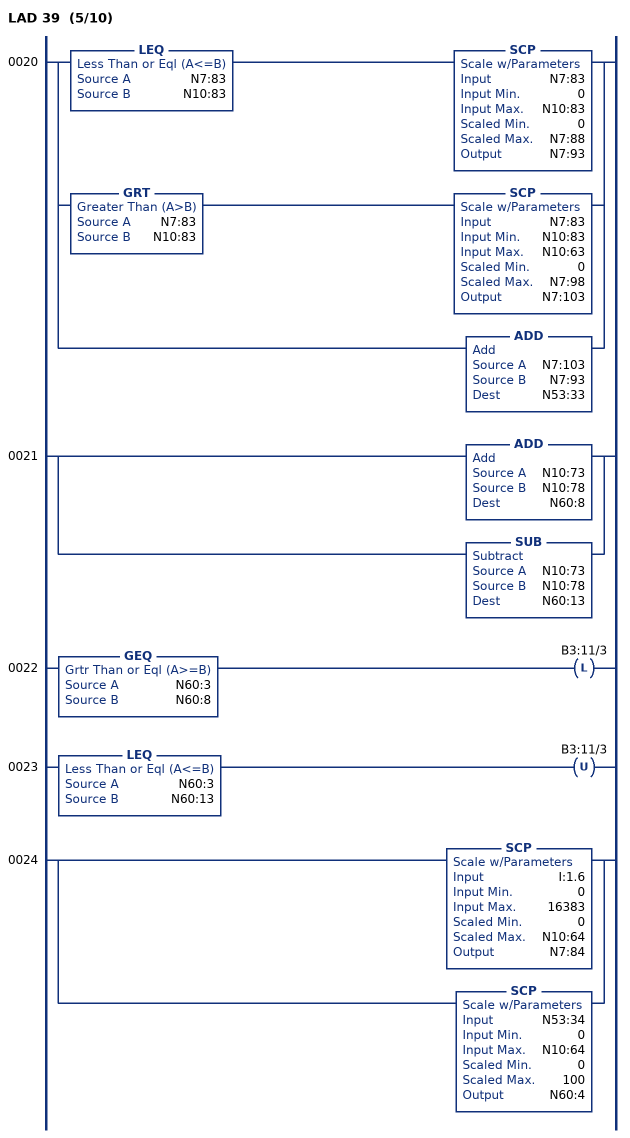
% Rung: 20 %
SOR BST LEQ N7:83 N10:83 SCP N7:83 0 N10:83 0 N7:88 N7:93 NXB GRT N7:83 N10:83 SCP N7:83 N10:83 N10:63 0 N7:98 N7:103 NXB ADD N7:103 N7:93 N53:33 BND EOR
% Rung: 21 %
SOR BST ADD N10:73 N10:78 N60:8 NXB SUB N10:73 N10:78 N60:13 BND EOR
% Rung: 22 %
SOR GEQ N60:3 N60:8 OTL B3:11/3 EOR
% Rung: 23 %
SOR LEQ N60:3 N60:13 OTU B3:11/3 EOR
% Rung: 24 %
SOR BST SCP I:1.6 0 16383 0 N10:64 N7:84 NXB SCP N53:34 0 N10:64 0 100 N60:4 BND EOR

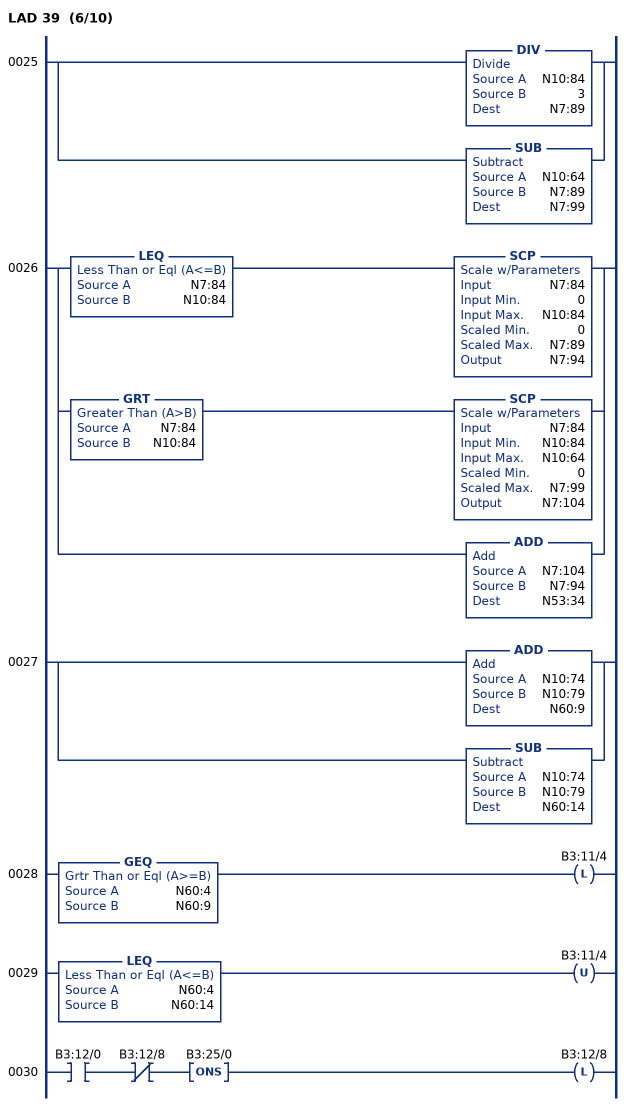
% Rung: 25 %
SOR BST DIV N10:84 3 N7:89 NXB SUB N10:64 N7:89 N7:99 BND EOR
% Rung: 26 %
SOR BST LEQ N7:84 N10:84 SCP N7:84 0 N10:84 0 N7:89 N7:94 NXB GRT N7:84 N10:84 SCP N7:84 N10:84 N10:64 0 N7:99 N7:104 NXB ADD N7:104 N7:94 N53:34 BND EOR
% Rung: 27 %
SOR BST ADD N10:74 N10:79 N60:9 NXB SUB N10:74 N10:79 N60:14 BND EOR
% Rung: 28 %
SOR GEQ N60:4 N60:9 OTL B3:11/4 EOR
% Rung: 29 %
SOR LEQ N60:4 N60:14 OTU B3:11/4 EOR
% Rung: 30 %
SOR XIC B3:12/0 XIO B3:12/8 OSR B3:25/0 OTL B3:12/8 EOR

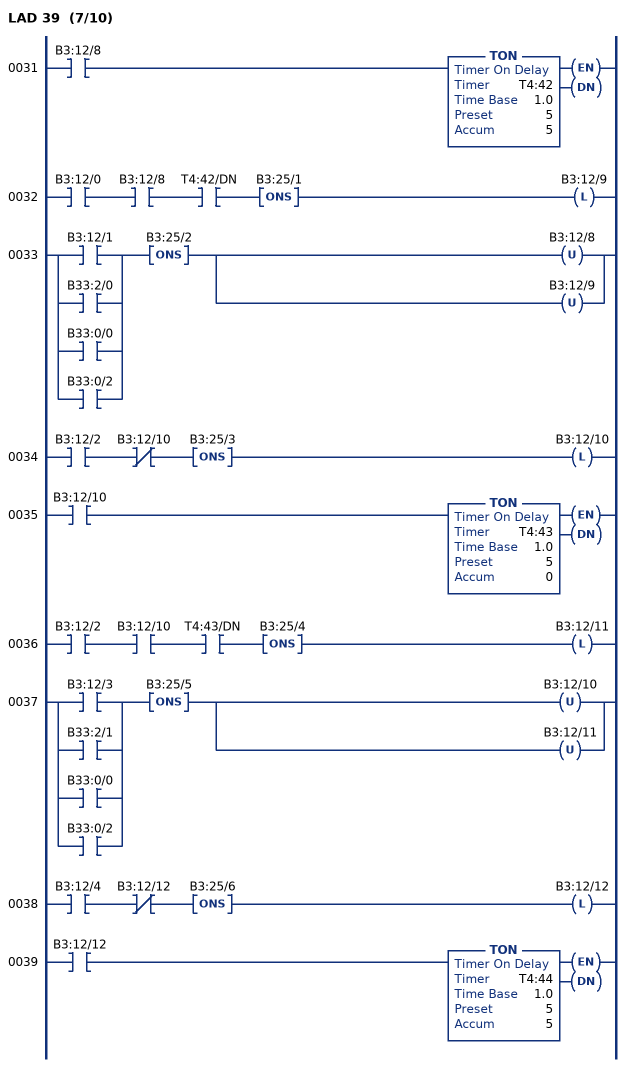
% Rung: 31 %
SOR XIC B3:12/8 TON T4:42 1.0 5 5 EOR
% Rung: 32 %
SOR XIC B3:12/0 XIC B3:12/8 XIC T4:42/DN OSR B3:25/1 OTL B3:12/9 EOR
% Rung: 33 %
SOR BST XIC B3:12/1 NXB XIC B33:2/0 NXB XIC B33:0/0 NXB XIC B33:0/2 BND OSR B3:25/2 BST OTU B3:12/8 NXB OTU B3:12/9 BND EOR
% Rung: 34 %
SOR XIC B3:12/2 XIO B3:12/10 OSR B3:25/3 OTL B3:12/10 EOR
% Rung: 35 %
SOR XIC B3:12/10 TON T4:43 1.0 5 0 EOR
% Rung: 36 %
SOR XIC B3:12/2 XIC B3:12/10 XIC T4:43/DN OSR B3:25/4 OTL B3:12/11 EOR
% Rung: 37 %
SOR BST XIC B3:12/3 NXB XIC B33:2/1 NXB XIC B33:0/0 NXB XIC B33:0/2 BND OSR B3:25/5 BST OTU B3:12/10 NXB OTU B3:12/11 BND EOR
% Rung: 38 %
SOR XIC B3:12/4 XIO B3:12/12 OSR B3:25/6 OTL B3:12/12 EOR
% Rung: 39 %
SOR XIC B3:12/12 TON T4:44 1.0 5 5 EOR

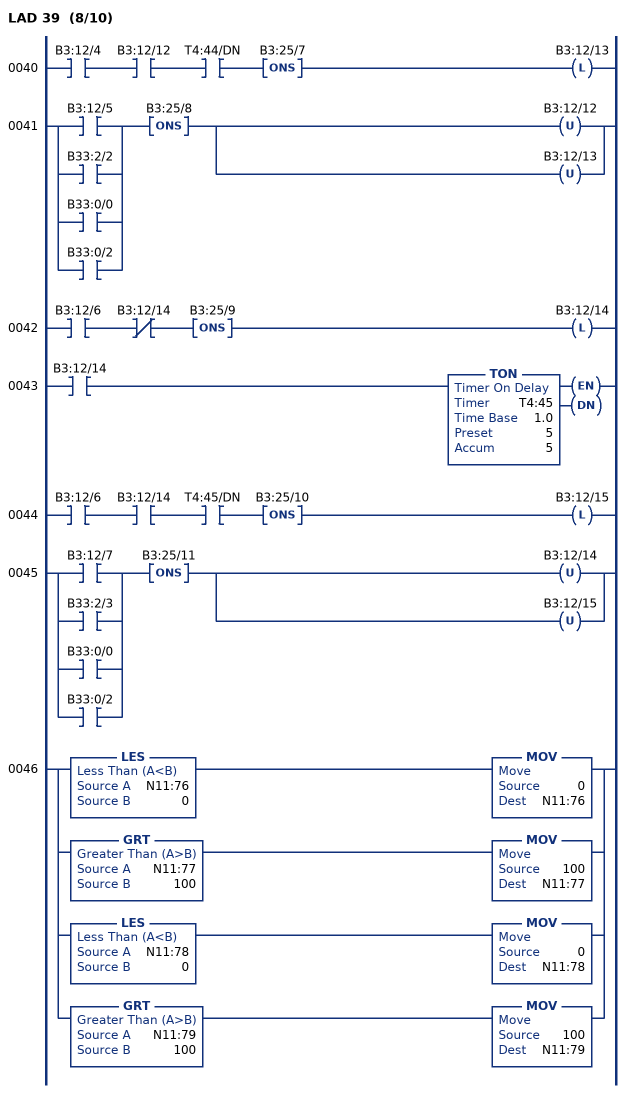
% Rung: 40 %
SOR XIC B3:12/4 XIC B3:12/12 XIC T4:44/DN OSR B3:25/7 OTL B3:12/13 EOR
% Rung: 41 %
SOR BST XIC B3:12/5 NXB XIC B33:2/2 NXB XIC B33:0/0 NXB XIC B33:0/2 BND OSR B3:25/8 BST OTU B3:12/12 NXB OTU B3:12/13 BND EOR
% Rung: 42 %
SOR XIC B3:12/6 XIO B3:12/14 OSR B3:25/9 OTL B3:12/14 EOR
% Rung: 43 %
SOR XIC B3:12/14 TON T4:45 1.0 5 5 EOR
% Rung: 44 %
SOR XIC B3:12/6 XIC B3:12/14 XIC T4:45/DN OSR B3:25/10 OTL B3:12/15 EOR
% Rung: 45 %
SOR BST XIC B3:12/7 NXB XIC B33:2/3 NXB XIC B33:0/0 NXB XIC B33:0/2 BND OSR B3:25/11 BST OTU B3:12/14 NXB OTU B3:12/15 BND EOR
% Rung: 46 %
SOR BST LES N11:76 0 MOV 0 N11:76 NXB GRT N11:77 100 MOV 100 N11:77 NXB LES N11:78 0 MOV 0 N11:78 NXB GRT N11:79 100 MOV 100 N11:79 BND EOR

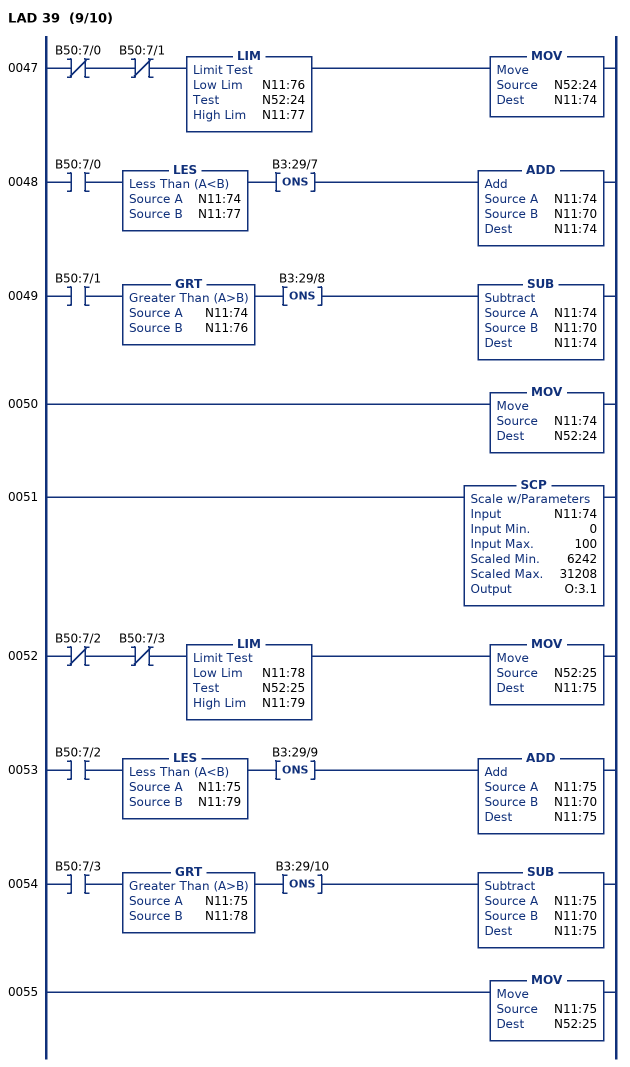
% Rung: 47 %
SOR XIO B50:7/0 XIO B50:7/1 LIM N11:76 N52:24 N11:77 MOV N52:24 N11:74 EOR
% Rung: 48 %
SOR XIC B50:7/0 LES N11:74 N11:77 OSR B3:29/7 ADD N11:74 N11:70 N11:74 EOR
% Rung: 49 %
SOR XIC B50:7/1 GRT N11:74 N11:76 OSR B3:29/8 SUB N11:74 N11:70 N11:74 EOR
% Rung: 50 %
SOR MOV N11:74 N52:24 EOR
% Rung: 51 %
SOR SCP N11:74 0 100 6242 31208 O:3.1 EOR
% Rung: 52 %
SOR XIO B50:7/2 XIO B50:7/3 LIM N11:78 N52:25 N11:79 MOV N52:25 N11:75 EOR
% Rung: 53 %
SOR XIC B50:7/2 LES N11:75 N11:79 OSR B3:29/9 ADD N11:75 N11:70 N11:75 EOR
% Rung: 54 %
SOR XIC B50:7/3 GRT N11:75 N11:78 OSR B3:29/10 SUB N11:75 N11:70 N11:75 EOR
% Rung: 55 %
SOR MOV N11:75 N52:25 EOR

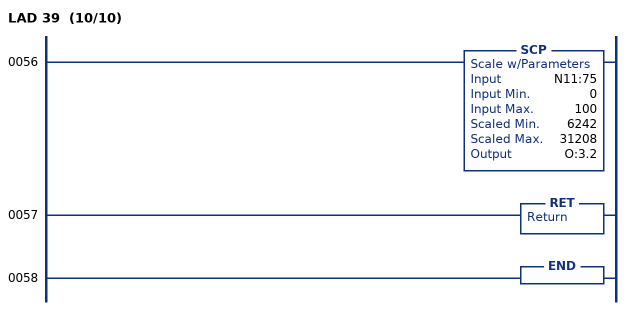
% Rung: 56 %
SOR SCP N11:75 0 100 6242 31208 O:3.2 EOR
% Rung: 57 %
SOR RET EOR
% Rung: 58 %
SOR END EOR

LADDER 40
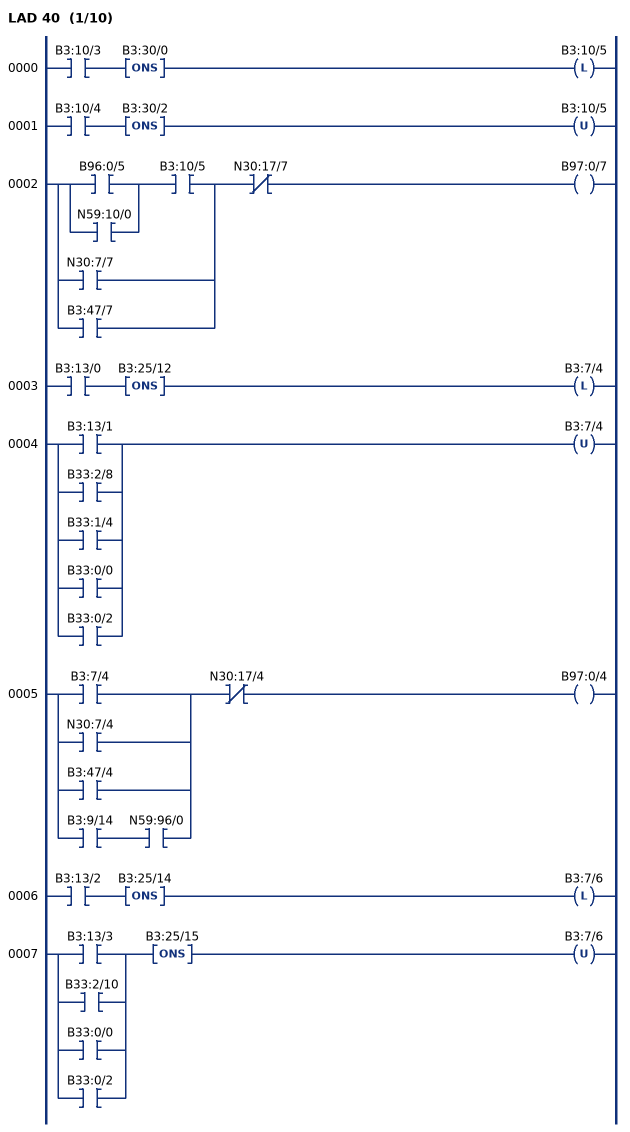
% Rung: 0 %
SOR XIC B3:10/3 OSR B3:30/0 OTL B3:10/5 EOR
% Rung: 1 %
SOR XIC B3:10/4 OSR B3:30/2 OTU B3:10/5 EOR
% Rung: 2 %
SOR BST BST XIC B96:0/5 NXB XIC N59:10/0 BND XIC B3:10/5 NXB XIC N30:7/7 NXB XIC B3:47/7 BND XIO N30:17/7 OTE B97:0/7 EOR
% Rung: 3 %
SOR XIC B3:13/0 OSR B3:25/12 OTL B3:7/4 EOR
% Rung: 4 %
SOR BST XIC B3:13/1 NXB XIC B33:2/8 NXB XIC B33:1/4 NXB XIC B33:0/0 NXB XIC B33:0/2 BND OTU B3:7/4 EOR
% Rung: 5 %
SOR BST XIC B3:7/4 NXB XIC N30:7/4 NXB XIC B3:47/4 NXB XIC B3:9/14 XIC N59:96/0 BND XIO N30:17/4 OTE B97:0/4 EOR
% Rung: 6 %
SOR XIC B3:13/2 OSR B3:25/14 OTL B3:7/6 EOR
% Rung: 7 %
SOR BST XIC B3:13/3 NXB XIC B33:2/10 NXB XIC B33:0/0 NXB XIC B33:0/2 BND OSR B3:25/15 OTU B3:7/6 EOR

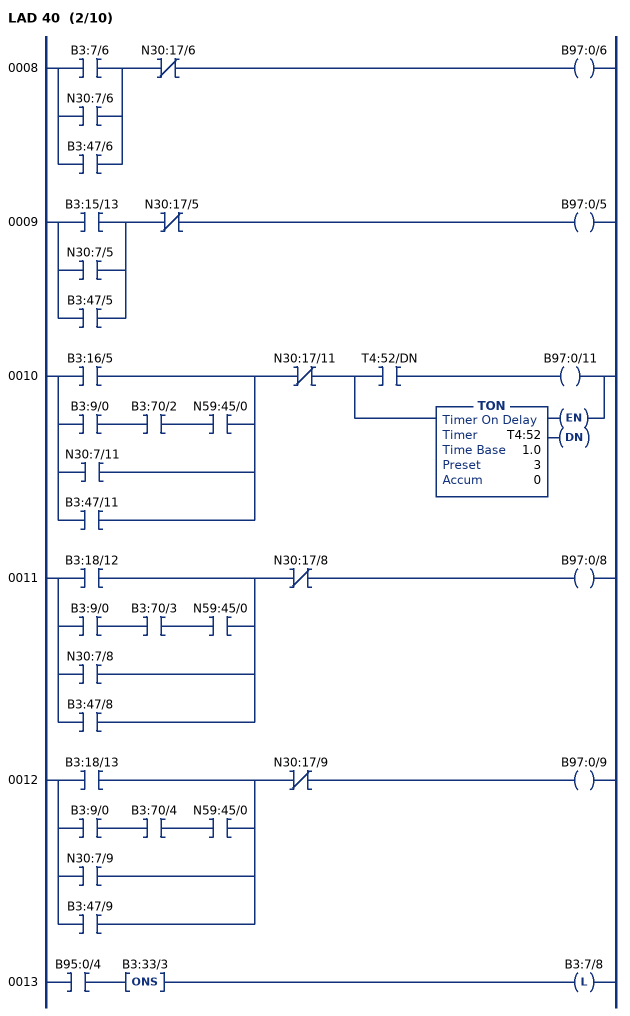
% Rung: 8 %
SOR BST XIC B3:7/6 NXB XIC N30:7/6 NXB XIC B3:47/6 BND XIO N30:17/6 OTE B97:0/6 EOR
% Rung: 9 %
SOR BST XIC B3:15/13 NXB XIC N30:7/5 NXB XIC B3:47/5 BND XIO N30:17/5 OTE B97:0/5 EOR
% Rung: 10 %
SOR BST XIC B3:16/5 NXB XIC B3:9/0 XIC B3:70/2 XIC N59:45/0 NXB XIC N30:7/11 NXB XIC B3:47/11 BND XIO N30:17/11 BST XIC T4:52/DN OTE B97:0/11 NXB TON T4:52 1.0 3 0 BND EOR
% Rung: 11 %
SOR BST XIC B3:18/12 NXB XIC B3:9/0 XIC B3:70/3 XIC N59:45/0 NXB XIC N30:7/8 NXB XIC B3:47/8 BND XIO N30:17/8 OTE B97:0/8 EOR
% Rung: 12 %
SOR BST XIC B3:18/13 NXB XIC B3:9/0 XIC B3:70/4 XIC N59:45/0 NXB XIC N30:7/9 NXB XIC B3:47/9 BND XIO N30:17/9 OTE B97:0/9 EOR
% Rung: 13 %
SOR XIC B95:0/4 OSR B3:33/3 OTL B3:7/8 EOR

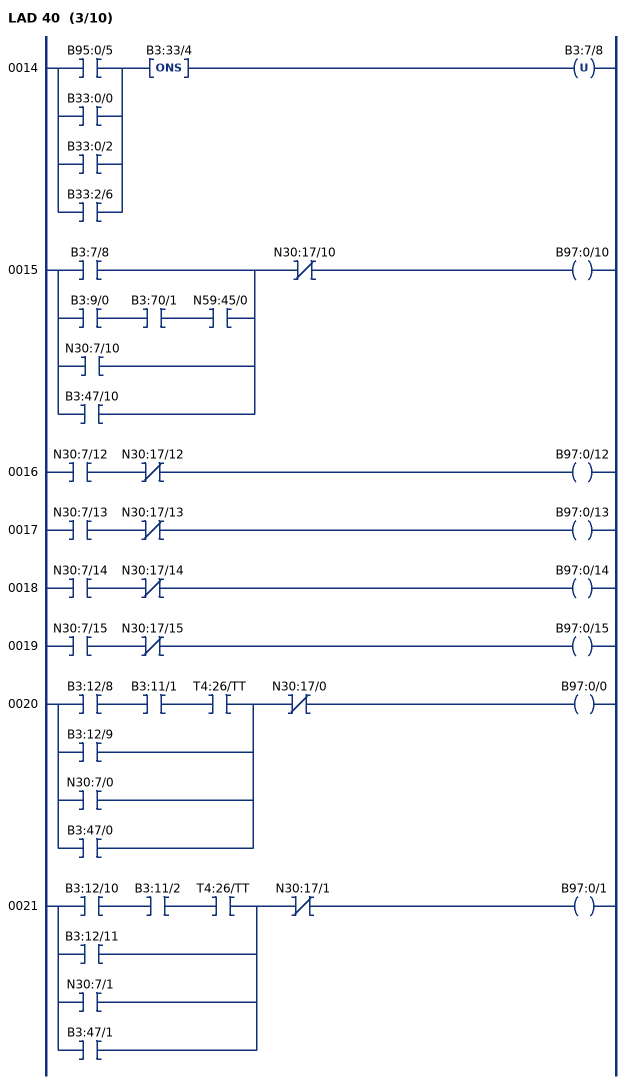
% Rung: 14 %
SOR BST XIC B95:0/5 NXB XIC B33:0/0 NXB XIC B33:0/2 NXB XIC B33:2/6 BND OSR B3:33/4 OTU B3:7/8 EOR
% Rung: 15 %
SOR BST XIC B3:7/8 NXB XIC B3:9/0 XIC B3:70/1 XIC N59:45/0 NXB XIC N30:7/10 NXB XIC B3:47/10 BND XIO N30:17/10 OTE B97:0/10 EOR
% Rung: 16 %
SOR XIC N30:7/12 XIO N30:17/12 OTE B97:0/12 EOR
% Rung: 17 %
SOR XIC N30:7/13 XIO N30:17/13 OTE B97:0/13 EOR
% Rung: 18 %
SOR XIC N30:7/14 XIO N30:17/14 OTE B97:0/14 EOR
% Rung: 19 %
SOR XIC N30:7/15 XIO N30:17/15 OTE B97:0/15 EOR
% Rung: 20 %
SOR BST BST XIC B3:12/8 XIC B3:11/1 XIC T4:26/TT NXB XIC B3:12/9 BND NXB XIC N30:7/0 NXB XIC B3:47/0 BND XIO N30:17/0 OTE B97:0/0 EOR
% Rung: 21 %
SOR BST BST XIC B3:12/10 XIC B3:11/2 XIC T4:26/TT NXB XIC B3:12/11 BND NXB XIC N30:7/1 NXB XIC B3:47/1 BND XIO N30:17/1 OTE B97:0/1 EOR

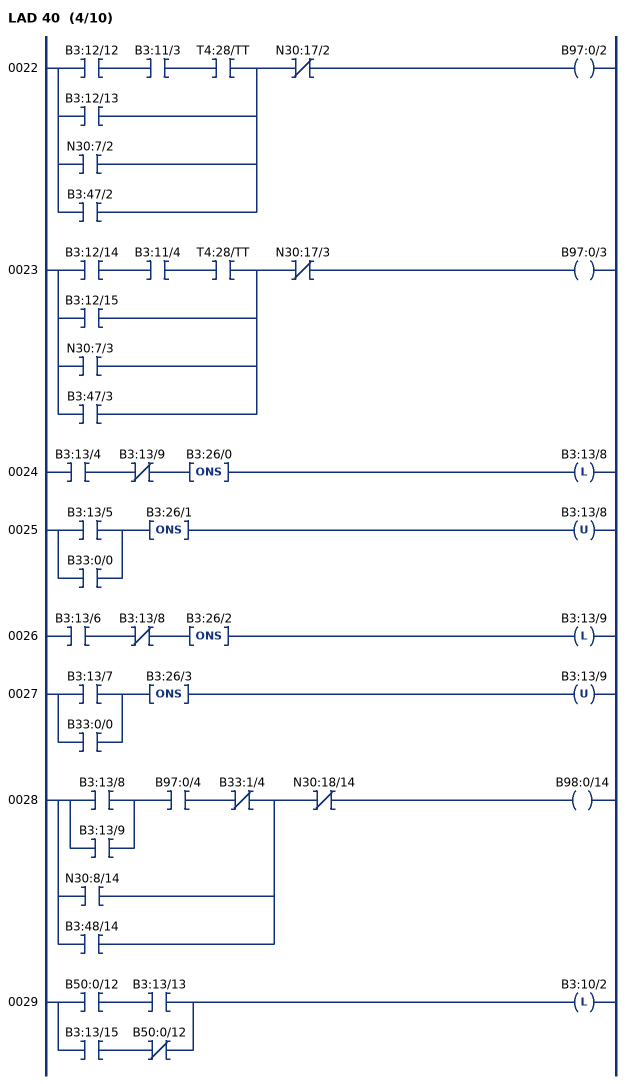
% Rung: 22 %
SOR BST BST XIC B3:12/12 XIC B3:11/3 XIC T4:28/TT NXB XIC B3:12/13 BND NXB XIC N30:7/2 NXB XIC B3:47/2 BND XIO N30:17/2 OTE B97:0/2 EOR
% Rung: 23 %
SOR BST BST XIC B3:12/14 XIC B3:11/4 XIC T4:28/TT NXB XIC B3:12/15 BND NXB XIC N30:7/3 NXB XIC B3:47/3 BND XIO N30:17/3 OTE B97:0/3 EOR
% Rung: 24 %
SOR XIC B3:13/4 XIO B3:13/9 OSR B3:26/0 OTL B3:13/8 EOR
% Rung: 25 %
SOR BST XIC B3:13/5 NXB XIC B33:0/0 BND OSR B3:26/1 OTU B3:13/8 EOR
% Rung: 26 %
SOR XIC B3:13/6 XIO B3:13/8 OSR B3:26/2 OTL B3:13/9 EOR
% Rung: 27 %
SOR BST XIC B3:13/7 NXB XIC B33:0/0 BND OSR B3:26/3 OTU B3:13/9 EOR
% Rung: 28 %
SOR BST BST XIC B3:13/8 NXB XIC B3:13/9 BND XIC B97:0/4 XIO B33:1/4 NXB XIC N30:8/14 NXB XIC B3:48/14 BND XIO N30:18/14 OTE B98:0/14 EOR
% Rung: 29 %
SOR BST XIC B50:0/12 XIC B3:13/13 NXB XIC B3:13/15 XIO B50:0/12 BND OTL B3:10/2 EOR

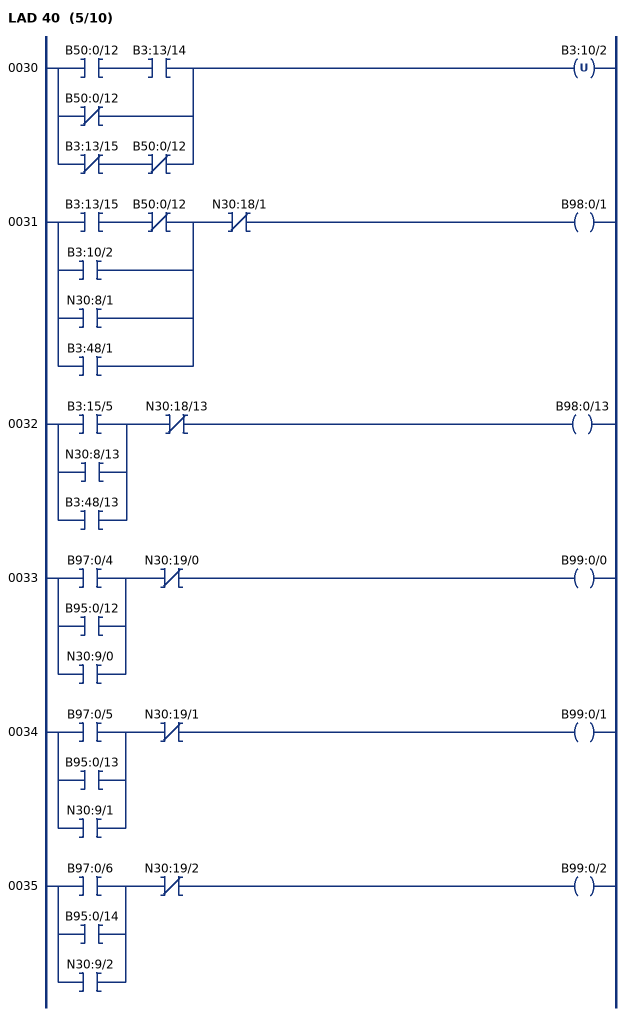
% Rung: 30 %
SOR BST XIC B50:0/12 XIC B3:13/14 NXB XIO B50:0/12 NXB XIO B3:13/15 XIO B50:0/12 BND OTU B3:10/2 EOR
% Rung: 31 %
SOR BST BST XIC B3:13/15 XIO B50:0/12 NXB XIC B3:10/2 BND NXB XIC N30:8/1 NXB XIC B3:48/1 BND XIO N30:18/1 OTE B98:0/1 EOR
% Rung: 32 %
SOR BST XIC B3:15/5 NXB XIC N30:8/13 NXB XIC B3:48/13 BND XIO N30:18/13 OTE B98:0/13 EOR
% Rung: 33 %
SOR BST BST XIC B97:0/4 NXB XIC B95:0/12 BND NXB XIC N30:9/0 BND XIO N30:19/0 OTE B99:0/0 EOR
% Rung: 34 %
SOR BST BST XIC B97:0/5 NXB XIC B95:0/13 BND NXB XIC N30:9/1 BND XIO N30:19/1 OTE B99:0/1 EOR
% Rung: 35 %
SOR BST BST XIC B97:0/6 NXB XIC B95:0/14 BND NXB XIC N30:9/2 BND XIO N30:19/2 OTE B99:0/2 EOR

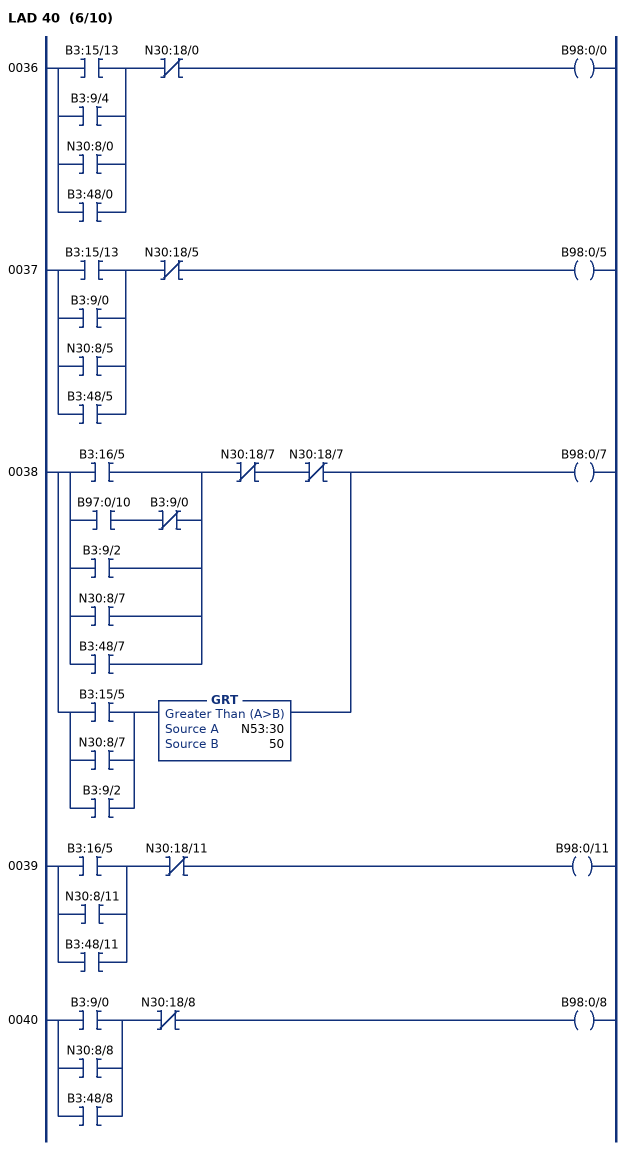
% Rung: 36 %
SOR BST XIC B3:15/13 NXB XIC B3:9/4 NXB XIC N30:8/0 NXB XIC B3:48/0 BND XIO N30:18/0 OTE B98:0/0 EOR
% Rung: 37 %
SOR BST XIC B3:15/13 NXB XIC B3:9/0 NXB XIC N30:8/5 NXB XIC B3:48/5 BND XIO N30:18/5 OTE B98:0/5 EOR
% Rung: 38 %
SOR BST BST XIC B3:16/5 NXB XIC B97:0/10 XIO B3:9/0 NXB XIC B3:9/2 NXB XIC N30:8/7 NXB XIC B3:48/7 BND XIO N30:18/7 XIO N30:18/7 NXB BST XIC B3:15/5 NXB BST XIC N30:8/7 NXB XIC B3:9/2 BND BND GRT N53:30 50 BND OTE B98:0/7 EOR
% Rung: 39 %
SOR BST XIC B3:16/5 NXB XIC N30:8/11 NXB XIC B3:48/11 BND XIO N30:18/11 OTE B98:0/11 EOR
% Rung: 40 %
SOR BST XIC B3:9/0 NXB XIC N30:8/8 NXB XIC B3:48/8 BND XIO N30:18/8 OTE B98:0/8 EOR

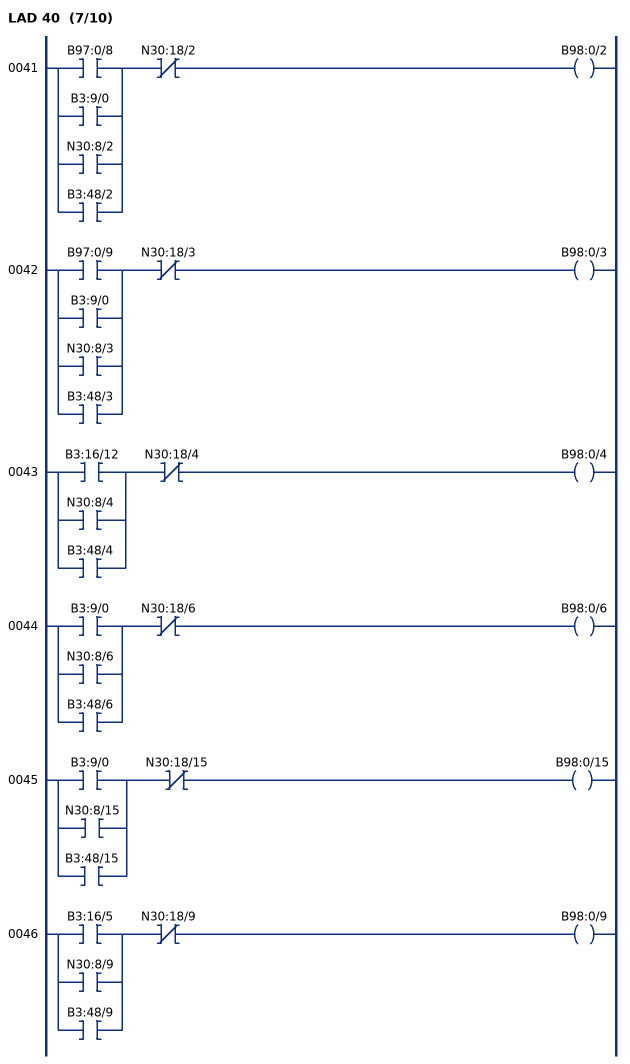
% Rung: 41 %
SOR BST XIC B97:0/8 NXB XIC B3:9/0 NXB XIC N30:8/2 NXB XIC B3:48/2 BND XIO N30:18/2 OTE B98:0/2 EOR
% Rung: 42 %
SOR BST XIC B97:0/9 NXB XIC B3:9/0 NXB XIC N30:8/3 NXB XIC B3:48/3 BND XIO N30:18/3 OTE B98:0/3 EOR
% Rung: 43 %
SOR BST XIC B3:16/12 NXB XIC N30:8/4 NXB XIC B3:48/4 BND XIO N30:18/4 OTE B98:0/4 EOR
% Rung: 44 %
SOR BST XIC B3:9/0 NXB XIC N30:8/6 NXB XIC B3:48/6 BND XIO N30:18/6 OTE B98:0/6 EOR
% Rung: 45 %
SOR BST XIC B3:9/0 NXB XIC N30:8/15 NXB XIC B3:48/15 BND XIO N30:18/15 OTE B98:0/15 EOR
% Rung: 46 %
SOR BST XIC B3:16/5 NXB XIC N30:8/9 NXB XIC B3:48/9 BND XIO N30:18/9 OTE B98:0/9 EOR

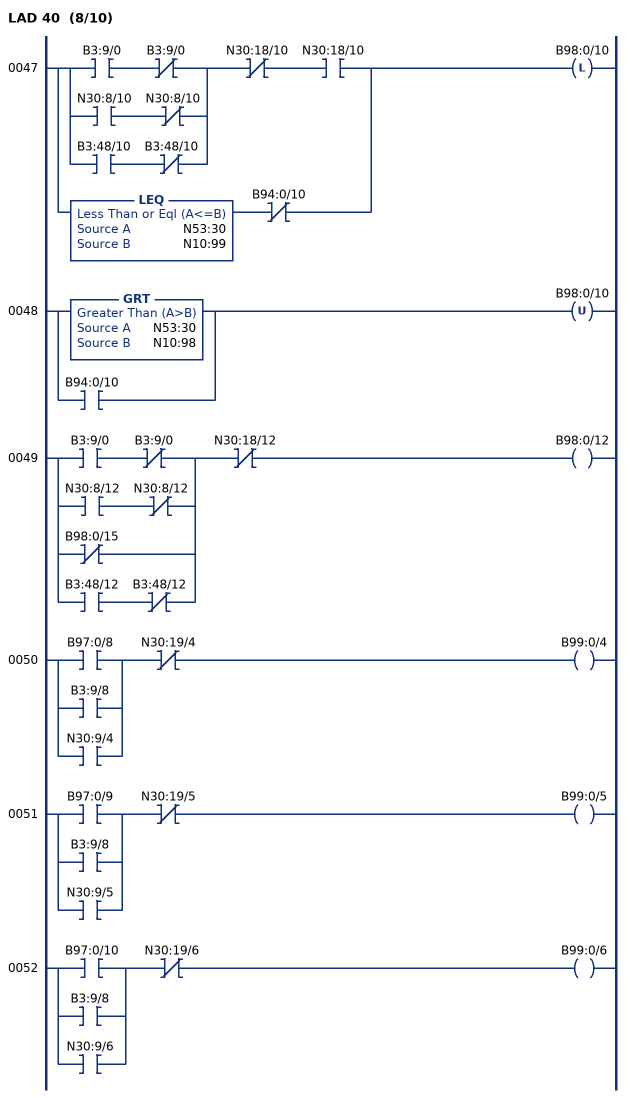
% Rung: 47 %
SOR BST BST XIC B3:9/0 XIO B3:9/0 NXB XIC N30:8/10 XIO N30:8/10 NXB XIC B3:48/10 XIO B3:48/10 BND XIO N30:18/10 XIC N30:18/10 NXB LEQ N53:30 N10:99 XIO B94:0/10 BND OTL B98:0/10 EOR
% Rung: 48 %
SOR BST GRT N53:30 N10:98 NXB XIC B94:0/10 BND OTU B98:0/10 EOR
% Rung: 49 %
SOR BST XIC B3:9/0 XIO B3:9/0 NXB XIC N30:8/12 XIO N30:8/12 NXB XIO B98:0/15 NXB XIC B3:48/12 XIO B3:48/12 BND XIO N30:18/12 OTE B98:0/12 EOR
% Rung: 50 %
SOR BST XIC B97:0/8 NXB XIC B3:9/8 NXB XIC N30:9/4 BND XIO N30:19/4 OTE B99:0/4 EOR
% Rung: 51 %
SOR BST XIC B97:0/9 NXB XIC B3:9/8 NXB XIC N30:9/5 BND XIO N30:19/5 OTE B99:0/5 EOR
% Rung: 52 %
SOR BST XIC B97:0/10 NXB XIC B3:9/8 NXB XIC N30:9/6 BND XIO N30:19/6 OTE B99:0/6 EOR

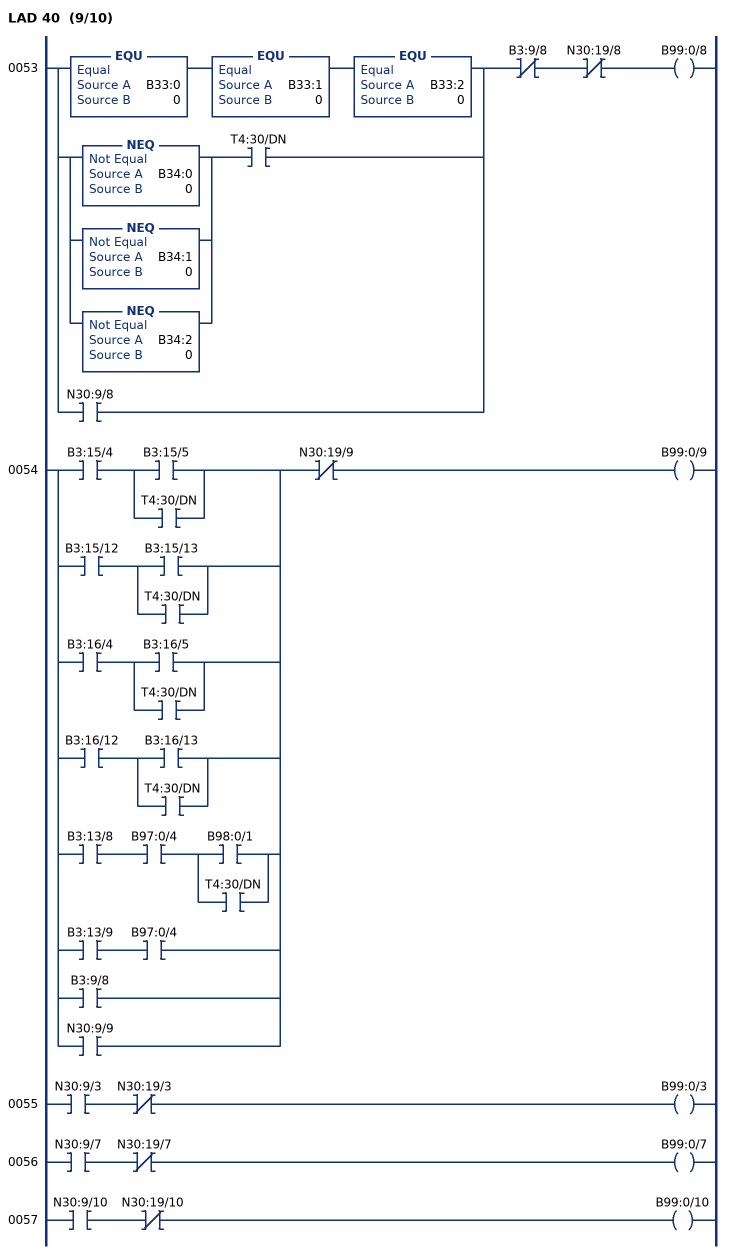
% Rung: 53 %
SOR BST EQU B33:0 0 EQU B33:1 0 EQU B33:2 0 NXB BST NEQ B34:0 0 NXB NEQ B34:1 0 NXB NEQ B34:2 0 BND XIC T4:30/DN NXB XIC N30:9/8 BND XIO B3:9/8 XIO N30:19/8 OTE B99:0/8 EOR
% Rung: 54 %
SOR BST XIC B3:15/4 BST XIC B3:15/5 NXB XIC T4:30/DN BND NXB XIC B3:15/12 BST XIC B3:15/13 NXB XIC T4:30/DN BND NXB XIC B3:16/4 BST XIC B3:16/5 NXB XIC T4:30/DN BND NXB XIC B3:16/12 BST XIC B3:16/13 NXB XIC T4:30/DN BND NXB XIC B3:13/8 XIC B97:0/4 BST XIC B98:0/1 NXB XIC T4:30/DN BND NXB XIC B3:13/9 XIC B97:0/4 NXB XIC B3:9/8 NXB XIC N30:9/9 BND XIO N30:19/9 OTE B99:0/9 EOR
% Rung: 55 %
SOR XIC N30:9/3 XIO N30:19/3 OTE B99:0/3 EOR
% Rung: 56 %
SOR XIC N30:9/7 XIO N30:19/7 OTE B99:0/7 EOR
% Rung: 57 %
SOR XIC N30:9/10 XIO N30:19/10 OTE B99:0/10 EOR

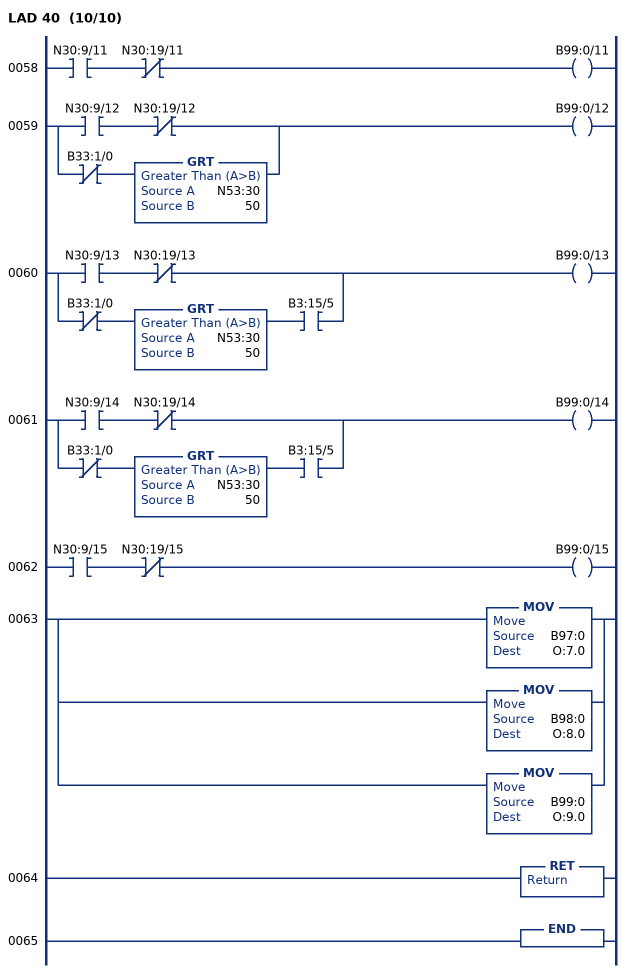
% Rung: 58 %
SOR XIC N30:9/11 XIO N30:19/11 OTE B99:0/11 EOR
% Rung: 59 %
SOR BST XIC N30:9/12 XIO N30:19/12 NXB XIO B33:1/0 GRT N53:30 50 BND OTE B99:0/12 EOR
% Rung: 60 %
SOR BST XIC N30:9/13 XIO N30:19/13 NXB XIO B33:1/0 GRT N53:30 50 XIC B3:15/5 BND OTE B99:0/13 EOR
% Rung: 61 %
SOR BST XIC N30:9/14 XIO N30:19/14 NXB XIO B33:1/0 GRT N53:30 50 XIC B3:15/5 BND OTE B99:0/14 EOR
% Rung: 62 %
SOR XIC N30:9/15 XIO N30:19/15 OTE B99:0/15 EOR
% Rung: 63 %
SOR BST MOV B97:0 O:7.0 NXB MOV B98:0 O:8.0 NXB MOV B99:0 O:9.0 BND EOR
% Rung: 64 %
SOR RET EOR
% Rung: 65 %
SOR END EOR

LADDER 50
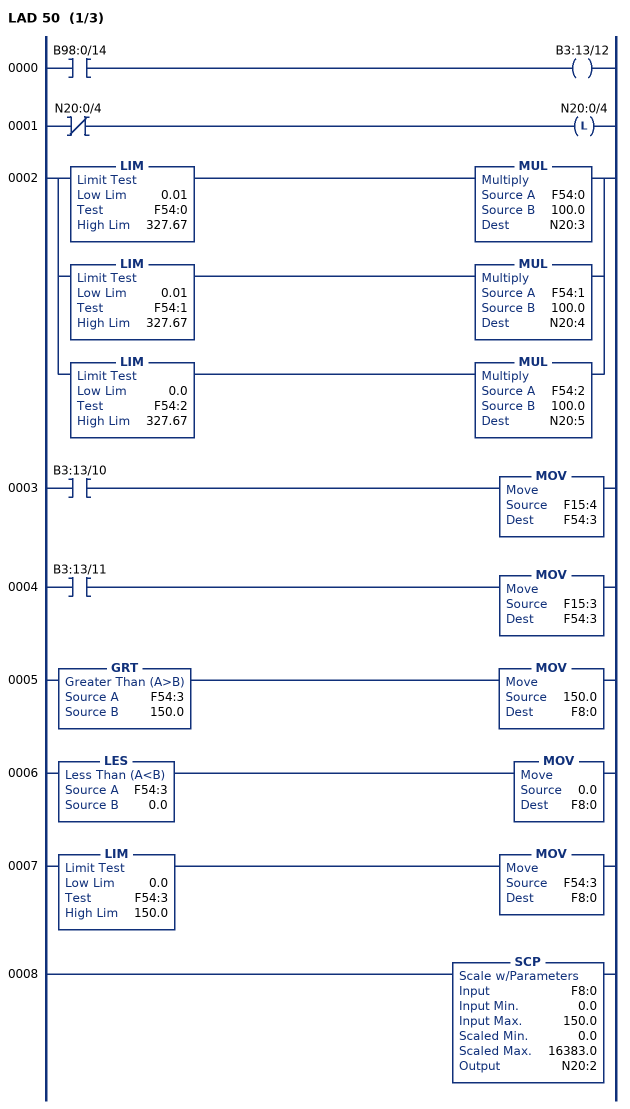
% Rung: 0 %
SOR XIC B98:0/14 OTE B3:13/12 EOR
% Rung: 1 %
SOR XIO N20:0/4 OTL N20:0/4 EOR
% Rung: 2 %
SOR BST LIM 0.01 F54:0 327.67 MUL F54:0 100.0 N20:3 NXB LIM 0.01 F54:1 327.67 MUL F54:1 100.0 N20:4 NXB LIM 0.0 F54:2 327.67 MUL F54:2 100.0 N20:5 BND EOR
% Rung: 3 %
SOR XIC B3:13/10 MOV F15:4 F54:3 EOR
% Rung: 4 %
SOR XIC B3:13/11 MOV F15:3 F54:3 EOR
% Rung: 5 %
SOR GRT F54:3 150.0 MOV 150.0 F8:0 EOR
% Rung: 6 %
SOR LES F54:3 0.0 MOV 0.0 F8:0 EOR
% Rung: 7 %
SOR LIM 0.0 F54:3 150.0 MOV F54:3 F8:0 EOR
% Rung: 8 %
SOR SCP F8:0 0.0 150.0 0.0 16383.0 N20:2 EOR

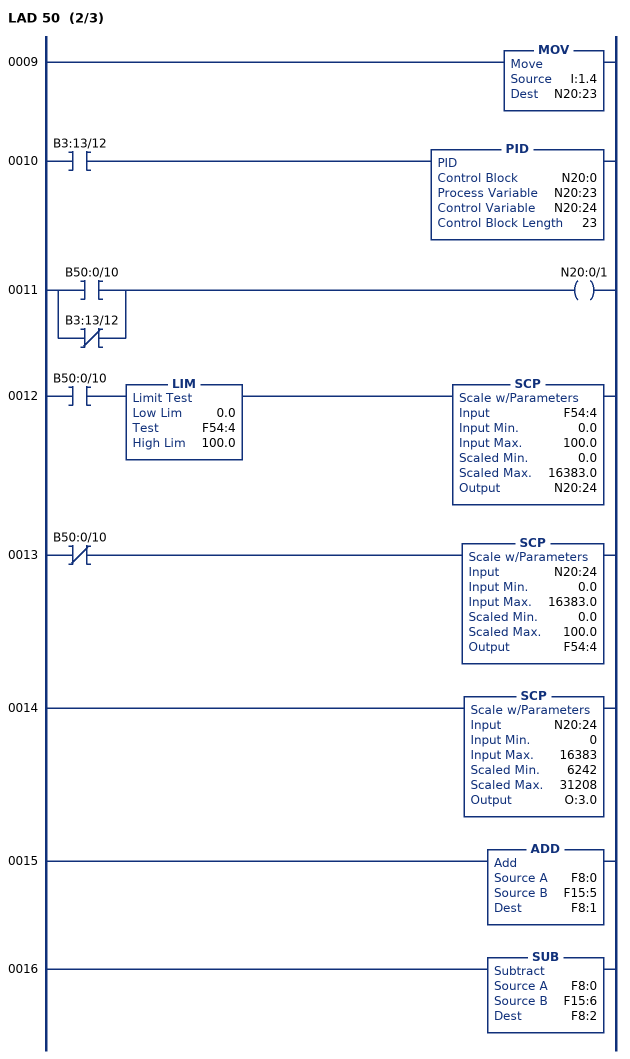
% Rung: 9 %
SOR MOV I:1.4 N20:23 EOR
% Rung: 10 %
SOR XIC B3:13/12 PID N20:0 N20:23 N20:24 23 EOR
% Rung: 11 %
SOR BST XIC B50:0/10 NXB XIO B3:13/12 BND OTE N20:0/1 EOR
% Rung: 12 %
SOR XIC B50:0/10 LIM 0.0 F54:4 100.0 SCP F54:4 0.0 100.0 0.0 16383.0 N20:24 EOR
% Rung: 13 %
SOR XIO B50:0/10 SCP N20:24 0.0 16383.0 0.0 100.0 F54:4 EOR
% Rung: 14 %
SOR SCP N20:24 0 16383 6242 31208 O:3.0 EOR
% Rung: 15 %
SOR ADD F8:0 F15:5 F8:1 EOR
% Rung: 16 %
SOR SUB F8:0 F15:6 F8:2 EOR

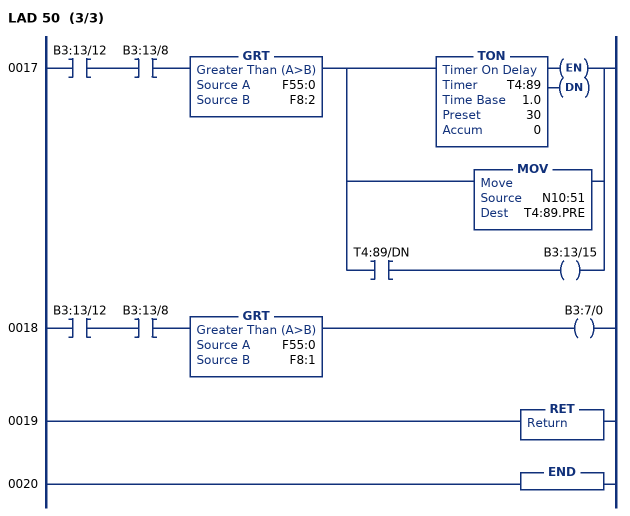
% Rung: 17 %
SOR XIC B3:13/12 XIC B3:13/8 GRT F55:0 F8:2 BST TON T4:89 1.0 30 0 NXB MOV N10:51 T4:89.PRE NXB XIC T4:89/DN OTE B3:13/15 BND EOR
% Rung: 18 %
SOR XIC B3:13/12 XIC B3:13/8 GRT F55:0 F8:1 OTE B3:7/0 EOR
% Rung: 19 %
SOR RET EOR
% Rung: 20 %
SOR END EOR

LADDER 75
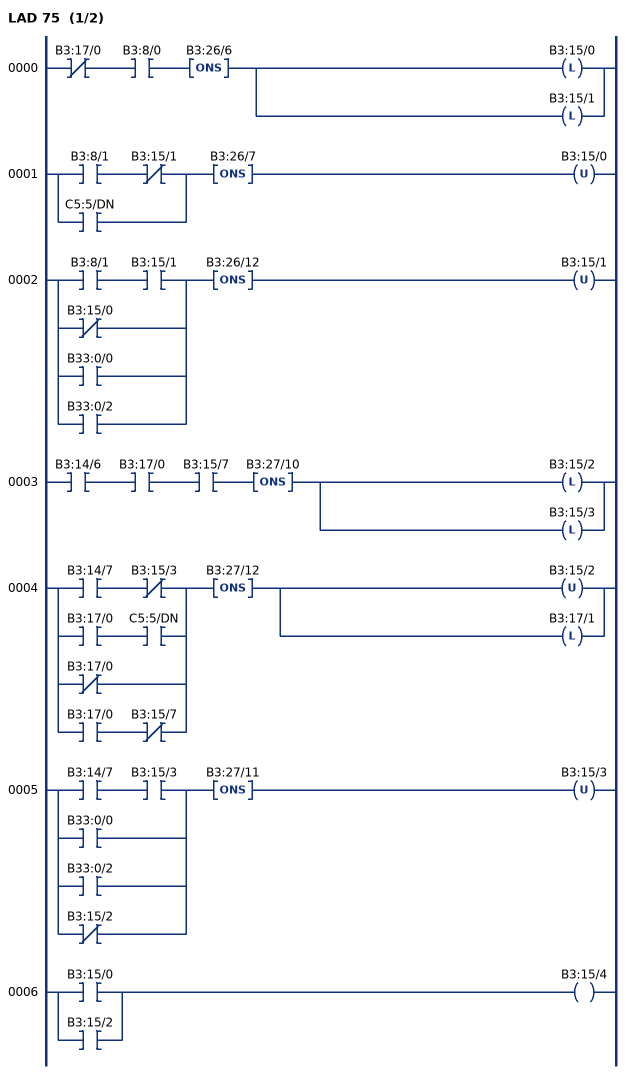
% Rung: 0 %
SOR XIO B3:17/0 XIC B3:8/0 OSR B3:26/6 BST OTL B3:15/0 NXB OTL B3:15/1 BND EOR
% Rung: 1 %
SOR BST XIC B3:8/1 XIO B3:15/1 NXB XIC C5:5/DN BND OSR B3:26/7 OTU B3:15/0 EOR
% Rung: 2 %
SOR BST XIC B3:8/1 XIC B3:15/1 NXB XIO B3:15/0 NXB XIC B33:0/0 NXB XIC B33:0/2 BND OSR B3:26/12 OTU B3:15/1 EOR
% Rung: 3 %
SOR XIC B3:14/6 XIC B3:17/0 XIC B3:15/7 OSR B3:27/10 BST OTL B3:15/2 NXB OTL B3:15/3 BND EOR
% Rung: 4 %
SOR BST XIC B3:14/7 XIO B3:15/3 NXB XIC B3:17/0 XIC C5:5/DN NXB XIO B3:17/0 NXB XIC B3:17/0 XIO B3:15/7 BND OSR B3:27/12 BST OTU B3:15/2 NXB OTL B3:17/1 BND EOR
% Rung: 5 %
SOR BST XIC B3:14/7 XIC B3:15/3 NXB XIC B33:0/0 NXB XIC B33:0/2 NXB XIO B3:15/2 BND OSR B3:27/11 OTU B3:15/3 EOR
% Rung: 6 %
SOR BST XIC B3:15/0 NXB XIC B3:15/2 BND OTE B3:15/4 EOR

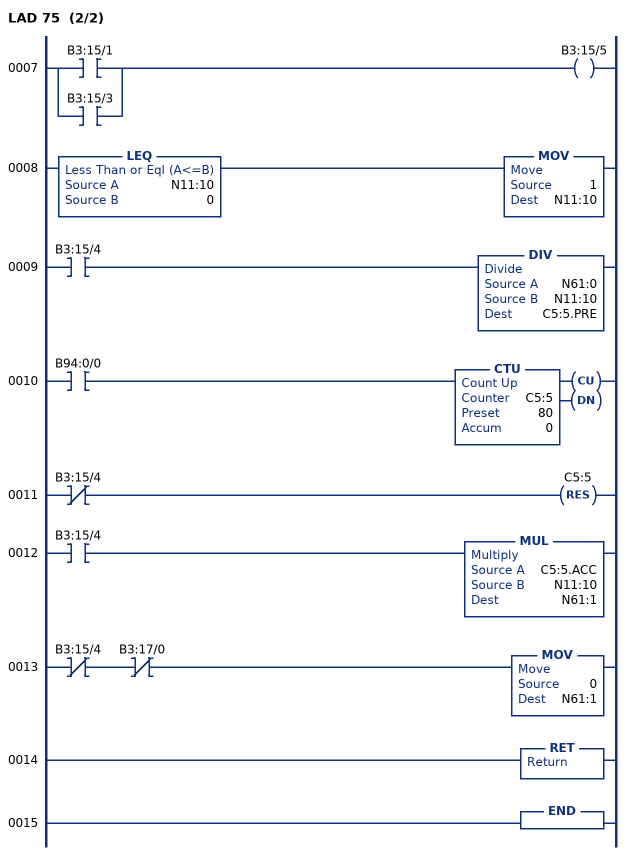
% Rung: 7 %
SOR BST XIC B3:15/1 NXB XIC B3:15/3 BND OTE B3:15/5 EOR
% Rung: 8 %
SOR LEQ N11:10 0 MOV 1 N11:10 EOR
% Rung: 9 %
SOR XIC B3:15/4 DIV N61:0 N11:10 C5:5.PRE EOR
% Rung: 10 %
SOR XIC B94:0/0 CTU C5:5 80 0 EOR
% Rung: 11 %
SOR XIO B3:15/4 RES C5:5 EOR
% Rung: 12 %
SOR XIC B3:15/4 MUL C5:5.ACC N11:10 N61:1 EOR
% Rung: 13 %
SOR XIO B3:15/4 XIO B3:17/0 MOV 0 N61:1 EOR
% Rung: 14 %
SOR RET EOR
% Rung: 15 %
SOR END EOR

LADDER 77
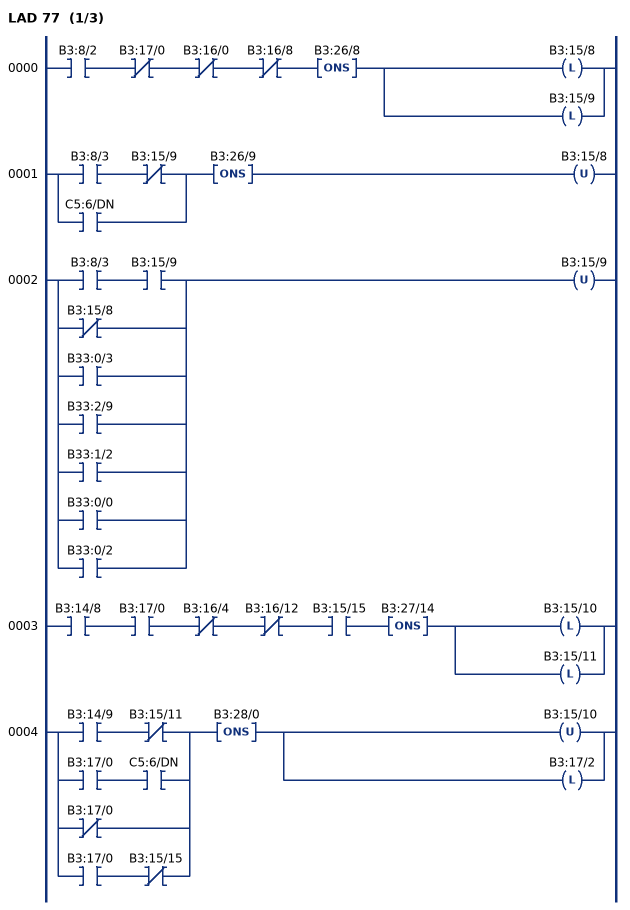
% Rung: 0 %
SOR XIC B3:8/2 XIO B3:17/0 XIO B3:16/0 XIO B3:16/8 OSR B3:26/8 BST OTL B3:15/8 NXB OTL B3:15/9 BND EOR
% Rung: 1 %
SOR BST XIC B3:8/3 XIO B3:15/9 NXB XIC C5:6/DN BND OSR B3:26/9 OTU B3:15/8 EOR
% Rung: 2 %
SOR BST XIC B3:8/3 XIC B3:15/9 NXB XIO B3:15/8 NXB XIC B33:0/3 NXB XIC B33:2/9 NXB XIC B33:1/2 NXB XIC B33:0/0 NXB XIC B33:0/2 BND OTU B3:15/9 EOR
% Rung: 3 %
SOR XIC B3:14/8 XIC B3:17/0 XIO B3:16/4 XIO B3:16/12 XIC B3:15/15 OSR B3:27/14 BST OTL B3:15/10 NXB OTL B3:15/11 BND EOR
% Rung: 4 %
SOR BST XIC B3:14/9 XIO B3:15/11 NXB XIC B3:17/0 XIC C5:6/DN NXB XIO B3:17/0 NXB XIC B3:17/0 XIO B3:15/15 BND OSR B3:28/0 BST OTU B3:15/10 NXB OTL B3:17/2 BND EOR

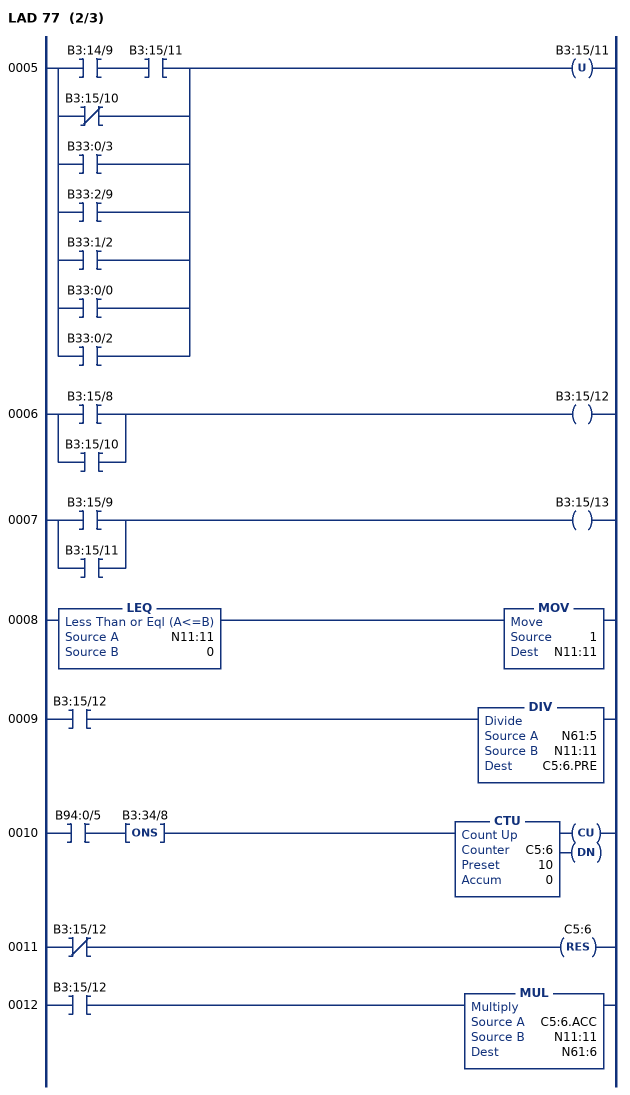
% Rung: 5 %
SOR BST XIC B3:14/9 XIC B3:15/11 NXB XIO B3:15/10 NXB XIC B33:0/3 NXB XIC B33:2/9 NXB XIC B33:1/2 NXB XIC B33:0/0 NXB XIC B33:0/2 BND OTU B3:15/11 EOR
% Rung: 6 %
SOR BST XIC B3:15/8 NXB XIC B3:15/10 BND OTE B3:15/12 EOR
% Rung: 7 %
SOR BST XIC B3:15/9 NXB XIC B3:15/11 BND OTE B3:15/13 EOR
% Rung: 8 %
SOR LEQ N11:11 0 MOV 1 N11:11 EOR
% Rung: 9 %
SOR XIC B3:15/12 DIV N61:5 N11:11 C5:6.PRE EOR
% Rung: 10 %
SOR XIC B94:0/5 OSR B3:34/8 CTU C5:6 10 0 EOR
% Rung: 11 %
SOR XIO B3:15/12 RES C5:6 EOR
% Rung: 12 %
SOR XIC B3:15/12 MUL C5:6.ACC N11:11 N61:6 EOR

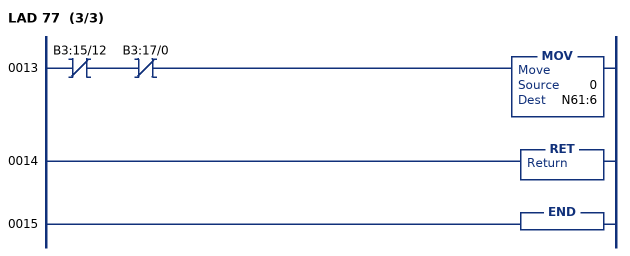
% Rung: 13 %
SOR XIO B3:15/12 XIO B3:17/0 MOV 0 N61:6 EOR
% Rung: 14 %
SOR RET EOR
% Rung: 15 %
SOR END EOR

LADDER 80
